{attribute addProperty BoxType "EPP1342-0001-0017"}
{attribute addProperty Id "A_0025_EPP1518_0002_0016EPP1518_1EB154A835444.25A_0026_EPP1518_0002_0017EPP1518_1EB154A835444.25A_0027_EPP1809_0021_0016EPP1809_248EAA3414618.25A_0028_EPP1809_0022_0016EPP1809_248EAA3414618.25A_0029_EPP1819_0021_0016EPP1819_248EAA3414618.25A_0030_EPP1819_0022_0016EPP1819_248EAA3414618.25A_0031_EPP1816_0003_0016EPP1816_8758F16324230.25A_0032_EPP1816_0008_0016EPP1816_C79E751722628.25A_0033_EPP1816_0008_0017EPP1816_C79E751722628.25A_0034_EPP1816_0008_0018EPP1816_8758F16324230.25A_0035_EPP1816_3008_0016EPP1816_F6DE3BA643454.25"}
{attribute addProperty CRC "3093405704"}
{attribute addProperty SizeInBites "2662"}
{attribute addProperty SizeInBytes "332.75"}
TYPE A_0024_EPP1342_0001_0017_B861A008 EXTENDS EPP1342_179A0949 :
STRUCT
	{attribute addProperty Name "A_0025_EPP1518_0002_0016"}
	A_0025_EPP1518_0002_0016 : EPP1518_1EB154A8;
	{attribute addProperty Name "A_0026_EPP1518_0002_0017"}
	A_0026_EPP1518_0002_0017 : EPP1518_1EB154A8;
	{attribute addProperty Name "A_0027_EPP1809_0021_0016"}
	A_0027_EPP1809_0021_0016 : EPP1809_248EAA34;
	{attribute addProperty Name "A_0028_EPP1809_0022_0016"}
	A_0028_EPP1809_0022_0016 : EPP1809_248EAA34;
	{attribute addProperty Name "A_0029_EPP1819_0021_0016"}
	A_0029_EPP1819_0021_0016 : EPP1819_248EAA34;
	{attribute addProperty Name "A_0030_EPP1819_0022_0016"}
	A_0030_EPP1819_0022_0016 : EPP1819_248EAA34;
	{attribute addProperty Name "A_0031_EPP1816_0003_0016"}
	A_0031_EPP1816_0003_0016 : EPP1816_8758F163;
	{attribute addProperty Name "A_0032_EPP1816_0008_0016"}
	A_0032_EPP1816_0008_0016 : EPP1816_C79E7517;
	{attribute addProperty Name "A_0033_EPP1816_0008_0017"}
	A_0033_EPP1816_0008_0017 : EPP1816_C79E7517;
	{attribute addProperty Name "A_0034_EPP1816_0008_0018"}
	A_0034_EPP1816_0008_0018 : EPP1816_8758F163;
	{attribute addProperty Name "A_0035_EPP1816_3008_0016"}
	A_0035_EPP1816_3008_0016 : EPP1816_F6DE3BA6;
END_STRUCT
END_TYPE

(* stored: Version 1.2.0.0, ProductVersion 3.1.4024.9
   DUT A_0024_EPP1342_0001_0017_B861A008: Id {e4fea851-5b52-41b8-9c45-4643ad181098} *)
